PROGRAM prgComEffIO
VAR
	fbCom		: FB_MqttCommunicator_v3;

END_VAR

fbCom(
	bConnect:= TRUE, 
	strAuthkey := 'DEV01673741737',
	sUserName:= '15132fb7-0bea-439b-8739-71b28de2c6f5' , 		
	sUserPassword:= '45379685-b2fb-4c09-8f03-19ad374f49d4',
	eSavePositionCertificate:= eSavePositionOnPLC.ePostionC, 
	bConnected=> , 
	bError=> , 
	hrErrorCode=> , 
	eConnectionState=> , 
	eErrorMessage_Out=> );

END_PROGRAM

(* stored: Version 1.1.0.1, ProductVersion 3.1.4024.12
   POU prgComEffIO: Id {7019f41b-2edd-476d-a8ca-340f2f7e1a91}, SpecialFunc None *)
